{attribute 'GeneratedUsingTerminal: EP9224-0037-0017'}
{attribute addProperty BoxType "EP9224-0037-0017"}
{attribute addProperty Id "StatusAT %I*Status_15ACD20111Current_UsAT %I*INT2Current_UpAT %I*INT2"}
{attribute addProperty CRC "242052069"}
{attribute addProperty Size "15"}
TYPE DPO_Inputs_Channel_0E6D6BE5 :
STRUCT
	{attribute addProperty Name "Status"}
	Status AT %I* : Status_15ACD201;
	{attribute addProperty Name "Current_Us"}
	Current_Us AT %I* : INT;
	{attribute addProperty Name "Current_Up"}
	Current_Up AT %I* : INT;
END_STRUCT
END_TYPE

(* stored: Version 1.2.0.0, ProductVersion 3.1.4024.9
   DUT DPO_Inputs_Channel_0E6D6BE5: Id {26c956ca-ffe7-46a9-b493-1bcb7797516f} *)
